INTERFACE ISignal EXTENDS IOut

METHOD Differentiate : IDifferentiable
VAR_INPUT
    deltaTime : Millisecond;
END_VAR
END_METHOD

METHOD Iir : IBaseSignal
VAR_INPUT
    decay : LREAL;
END_VAR
END_METHOD

METHOD Update : ISignal
VAR_INPUT
    value : LREAL;
END_VAR
END_METHOD

END_INTERFACE

(* stored: Version 1.1.0.1, ProductVersion 3.1.4024.12
   Itf ISignal: Id {83971406-8867-4284-ae5c-1ba41a8d6010}
   Method Differentiate: Id {87b91ba4-73cf-4951-a824-cab529987ebc}
   Method Iir: Id {dbc48f6e-24e3-46d0-8810-d8781ca3b879}
   Method Update: Id {96492a64-d485-4a2c-86bf-0390a7a3d226} *)
